# B&R Automation Studio project Laba2
Automation Studio 4.5.2.102

## Configuration labBR

CPU 4PP065.0571-P74, AutomationRuntime D4.52, Build 4.1.2, Vc V4.52.0, Safety 1.10

### Task classes (Cpu.sw)
```
Cyclic#1 (cycle 2000 us, tolerance 0 us):
  ncsdcctrl <- ncsdcctrl.prg
  DoorCtrl <- DoorCtrl.prg
Cyclic#7 (cycle 1000000 us, tolerance 1000000 us):
  LedCtrl <- LedCtrl.prg
DataObjects: Acp10sys, Arnc0sys
NcDataObjects: acp10etxen <- acp10etxen.dob, gmcipvar <- GmcIpUserConfig.gmcipvar.dob, gmcipfun <- GmcIpUserConfig.gmcipfun.dob, gmcipfub <- GmcIpUserConfig.gmcipfub.dob, gmcipubr <- GmcIpUserConfig.gmcipubr.dob, gmcipusm <- GmcIpUserConfig.gmcipusm.dob, gmcipui <- GmcIpUserConfig.gmcipui.dob, gmcipus <- GmcIpUserConfig.gmcipus.dob, gmcipuc <- GmcIpUserConfig.gmcipuc.dob, gmcipsys <- GmcIpConfig.gmcipsys.dob, gmciplbr <- GmcIpConfig.gmciplbr.dob, gmcipcbr <- GmcIpConfig.gmcipcbr.dob, gmciplsm <- GmcIpConfig.gmciplsm.dob, gmcipcsm <- GmcIpConfig.gmcipcsm.dob, gmcipcfg <- GmcIpConfig.gmcipcfg.dob, gmcipiec <- GmcIpConfig.gmcipiec.dob, gmciplog <- GmcIpConfig.gmciplog.dob, gmcipesm <- GmcIpConfig.gmcipesm.dob, gmcipmxd <- GmcIpConfig.gmcipmxd.dob, gmcipmx <- GmcIpConfig.gmcipmx.dob, gAxis01a <- gAxis01obj.gAxis01a.dob, gAxis01i <- gAxis01obj.gAxis01i.dob, gAxis02a <- gAxis02obj.gAxis02a.dob, gAxis02i <- gAxis02obj.gAxis02i.dob, gAxis03a <- gAxis03obj.gAxis03a.dob, gAxis03i <- gAxis03obj.gAxis03i.dob, gAxis04a <- gAxis04obj.gAxis04a.dob, gAxis04i <- gAxis04obj.gAxis04i.dob, gAxis05a <- gAxis05obj.gAxis05a.dob, gAxis05i <- gAxis05obj.gAxis05i.dob
Binaries: TCData, udbdef, iomap, sysconf, ashwac, ashwd, asfw, User, arconfig, Role, arnc0cfg, Arnc0map, Acp10map, acp10cfg
Libraries: Acp10man, Acp10par, NcGlobal, Acp10sdc, Arnc0man, DataObj, AsArLog, sys_lib, FileIO, AsArProf, AsMem, brsystem, runtime, astime, Acp10_MC, AsBrStr, X64Lib, GateCtrl, asieccon, powerlnk
```

### Hardware
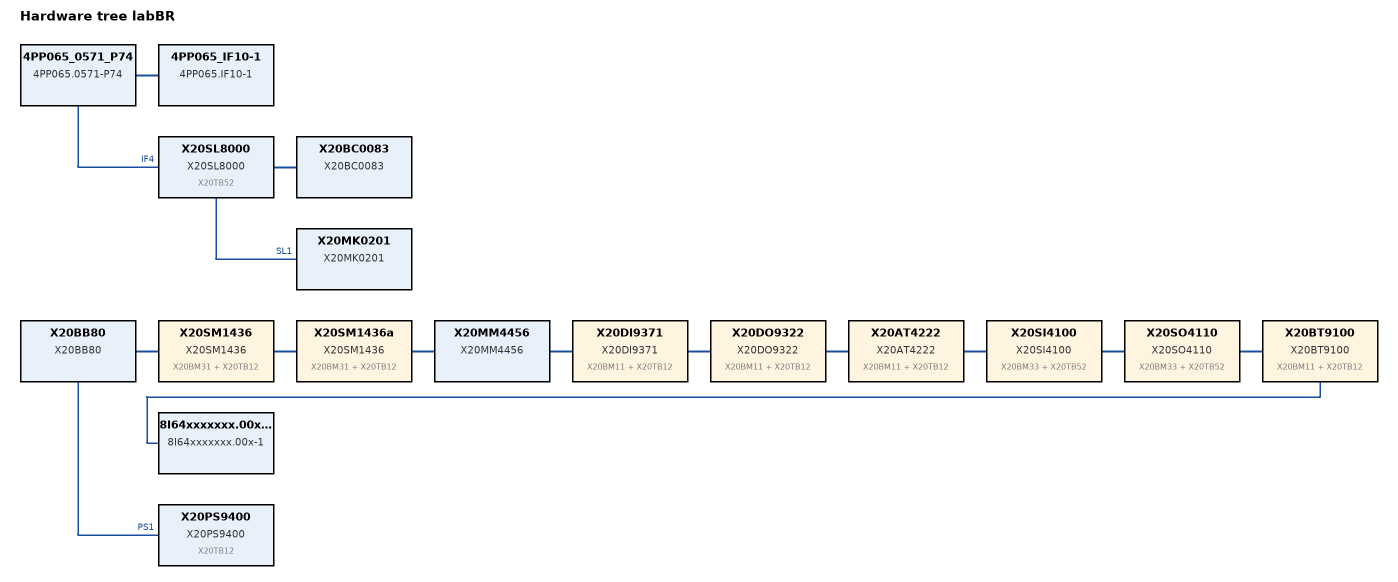
```
4PP065_0571_P74 : 4PP065.0571-P74 v1.1.2.0
  Connector IF4:
    EplInterfaceRedundant = 0
    EplEthInterfaceRedundant = 0
  Connector IF5:
    ActivateDevice = 1
    Mode = Manual
    InternetAddress = 10.1.1.13
    SubnetMask = 255.255.255.0
  ConfigurationID = DriveControl_SampleText
  TimerDeviceType = EPLX2X
  TimerDevice = 4PP065_0571_P74.IF4
  TaskClassIdleTime = 2000
  Cyclic1Duration = 2000
  Cyclic1Tolerance = 0
  Cyclic1Output = 1
  Cyclic2Duration = 20000
  Cyclic2Tolerance = 20000
  Cyclic3Duration = 50000
  Cyclic3Tolerance = 50000
  Cyclic4Duration = 100000
  Cyclic4Tolerance = 100000
  Cyclic5Duration = 200000
  Cyclic5Tolerance = 200000
  Cyclic6Duration = 500000
  Cyclic6Tolerance = 500000
  Cyclic7Duration = 1000000
  Cyclic7Tolerance = 1000000
  Cyclic8Duration = 10000
  Cyclic8Tolerance = 30000000
4PP065_IF10-1 : 4PP065.IF10-1 v1.0.3.0  [SS -> 4PP065_0571_P74.SS1]
8I64xxxxxxx.00x-1 : 8I64xxxxxxx.00x-1 v1.3.9.1  [X2X1 -> X20BT9100.X2X1 [Cable Type=X2XCable, Length=10, Version=1.0.0.2]]
  FunctionModel = Standard
  packedETAD = packed
  packedETI = packed
  packedCMDD = packed
  packedCMI = packed
  UNS = 220
  NCR = 10
  NSP = 890
  COS = 64
  RSC = 33000
X20AT4222 : X20AT4222 v1.2.3.0  [SS1 -> X20TB12e.SS; SL -> X20BM11c.SL1]
X20BB80 : X20BB80 v1.0.2.0
X20BC0083 : X20BC0083 v2.9.0.0  [PLK1 -> X20SL8000.PLK2 (NodeNumber=2) [Cable Type=PowerlinkCable, Length=10, Version=1.0.0.2]; SL -> X20BB80.SL1]
X20BM11 : X20BM11 v1.0.0.1  [X2X1 -> X20BM33a.X2X2]
X20BM11a : X20BM11 v1.0.0.1  [X2X1 -> X20MM4456.X2X2]
X20BM11b : X20BM11 v1.0.0.1  [X2X1 -> X20BM11a.X2X2]
X20BM11c : X20BM11 v1.0.0.1  [X2X1 -> X20BM11b.X2X2]
X20BM31 : X20BM31 v1.0.0.1  [X2X1 -> X20BB80.IF1]
X20BM31a : X20BM31 v1.0.0.1  [X2X1 -> X20BM31.X2X2]
X20BM33 : X20BM33 v1.0.0.4  [X2X1 -> X20BM11c.X2X2]
X20BM33a : X20BM33 v1.0.0.4  [X2X1 -> X20BM33.X2X2]
X20BT9100 : X20BT9100 v1.0.3.0  [SS1 -> X20TB12f.SS; SL -> X20BM11.SL1]
X20DI9371 : X20DI9371 v1.0.2.0  [SS1 -> X20TB12c.SS; SL -> X20BM11a.SL1]
X20DO9322 : X20DO9322 v1.0.3.0  [SS1 -> X20TB12d.SS; SL -> X20BM11b.SL1]
X20MK0201 : X20MK0201 v1.0.0.0  [SL -> X20SL8000.SL1]
X20MM4456 : X20MM4456 v1.1.5.0  [X2X1 -> X20BM31a.X2X2]
X20PS9400 : X20PS9400 v1.0.2.4  [SS1 -> X20TB12.SS; PS -> X20BB80.PS1]
X20SI4100 : X20SI4100 v1.10.1.1  [SS1 -> X20TB52.SS; SL -> X20BM33.SL1]
X20SL8000 : X20SL8000 v1.6.5.1  [PLK1 -> 4PP065_0571_P74.IF4 (NodeNumber=1) [Cable Type=PowerlinkCable, Length=10, Version=1.0.0.2]; PLK2 -> X20BC0083.PLK1 (NodeNumber=1) [Cable Type=PowerlinkCable, Length=10, Version=1.0.0.2]; SS1 -> X20TB52b.SS]
  SafeProject = SafeLOGIC-1
X20SM1436 : X20SM1436 v1.4.2.1  [SS1 -> X20TB12a.SS; SL -> X20BM31.SL1]
X20SM1436a : X20SM1436 v1.4.2.1  [SS1 -> X20TB12b.SS; SL -> X20BM31a.SL1]
X20SO4110 : X20SO4110 v1.10.1.1  [SS1 -> X20TB52a.SS; SL -> X20BM33a.SL1]
  SafeModuleID = 3
X20TB12 : X20TB12 v1.0.0.0
X20TB12a : X20TB12 v1.0.0.0
X20TB12b : X20TB12 v1.0.0.0
X20TB12c : X20TB12 v1.0.0.0
X20TB12d : X20TB12 v1.0.0.0
X20TB12e : X20TB12 v1.0.0.0
X20TB12f : X20TB12 v1.0.0.0
X20TB52 : X20TB52 v1.0.0.1
X20TB52a : X20TB52 v1.0.0.1
X20TB52b : X20TB52 v1.0.0.1
```

### IoMap.iom - 4PP065_0571_P74/IoMap.iom
```iecst
VAR_CONFIG
	::DoorCtrl:DoorBlock.s0 AT %IX."X20DI9371".DigitalInput02;
	::DoorCtrl:DoorBlock.s1 AT %IX."X20DI9371".DigitalInput03;
	::DoorCtrl:DoorBlock.s2 AT %IX."X20DI9371".DigitalInput04;
	::DoorCtrl:DoorBlock.s3 AT %IX."X20DI9371".DigitalInput05;
	::DoorCtrl:CMD AT %QW."8I64xxxxxxx.00x-1".CMDD_Output;
	::DoorCtrl:ETAD AT %IW."8I64xxxxxxx.00x-1".ETAD_Input;
	::DoorCtrl:Speed AT %QW."8I64xxxxxxx.00x-1".LFRD_Output;
END_VAR
```

## Logical view

Binary libraries used (declarations not repeated): operator, runtime, astime, AsIecCon, Acp10man, Acp10par, NcGlobal, Acp10sdc, Arnc0man, DataObj, AsArLog, sys_lib, FileIO, AsArProf, AsMem, brsystem, Acp10_MC, AsBrStr

### Global.var - Global variables
```iecst
VAR
	s1 : BOOL := FALSE;
	s2 : BOOL := FALSE;
	s3 : BOOL := FALSE;
	s0 : BOOL := FALSE;
END_VAR
```

### Package Logical/Libraries - Global libraries

### Library Logical/Libraries/X64Lib (ANSIC)

#### X64Lib.fun
```iecst
(********************************************************************
 * COPYRIGHT -- Microsoft
 ********************************************************************
 * Library: X64Lib
 * File: X64Lib.fun
 * Author: chuh
 * Created: April 02, 2015
 ********************************************************************
 * Functions and function blocks of library X64Lib
 ********************************************************************)

FUNCTION_BLOCK FBX64Inverter (*X64 Acopos Inverter Control Lib*) (*$GROUP=User*)
	VAR_INPUT
		enable : BOOL;
		ETAD_Input : UINT;
	END_VAR
	VAR_OUTPUT
		CMDD_Output : UINT;
	END_VAR
	VAR
		sex : UINT;
	END_VAR
END_FUNCTION_BLOCK
```

#### FBX64Inverter.c
```c
/********************************************************************
 * COPYRIGHT -- Microsoft
 ********************************************************************
 * Library: X64Lib
 * File: FBX64Inverter.c
 * Author: chuh
 * Created: April 02, 2015
 ********************************************************************
 * Implementation of library X64Lib
 ********************************************************************/

#include <bur/plctypes.h>
#ifdef __cplusplus
	extern "C"
	{
#endif

	#include "X64Lib.h"

#ifdef __cplusplus
	};
#endif

//***************Объявление списка состояний частотника ? ********************
#define	ACPIX64_STATE_NOT_READY_TO_SWITCH_ON	0x0000 /* */
#define	ACPIX64_STATE_SWITCH_ON_DISABLED		0x0040 /* */
#define	ACPIX64_STATE_READY_TO_SWITCH_ON		0x0064 /* */
#define	ACPIX64_STATE_SWITCHED_ON				0x0021 /* */
#define	ACPIX64_STATE_OPERATION_ENABLED			0x0027 /* */
#define	ACPIX64_STATE_QUICK_STOP_ACTIVE			0x0007/* */
#define	ACPIX64_STATE_MALFUNCTION				0x0008/* */

#define	ACPIX64_CMD_DISABLE_VOLTAGE				0x0000/* */
#define	ACPIX64_CMD_SHUTDOWN					0x0006/* */
#define	ACPIX64_CMD_SWITCH_ON					0x0006/* */
#define	ACPIX64_CMD_ENABLE_OPERATION			0x000F/* */
#define ACPIX64_CMD_GO                          0x0007
#define	ACPIX64_CMD_FAULT_RESET					0x0080/* */

/* X64 Acopos Inverter Control Lib */
void FBX64Inverter(struct FBX64Inverter* inst)
{
	UINT MSK;			//Переменная для хранения входа после наложения ма
	MSK = inst->ETAD_Input & 0x006F;
	inst->sex = MSK;/* */ // маска на значащую информацию статуса частотника
	if(!inst->enable){
		inst->CMDD_Output = ACPIX64_CMD_DISABLE_VOLTAGE;		//	 Отключаем питание с двигателя насоса
	} else {
		switch(MSK)
		{
			case ACPIX64_STATE_SWITCH_ON_DISABLED:		inst->CMDD_Output = ACPIX64_CMD_SHUTDOWN;				break;
			case ACPIX64_STATE_READY_TO_SWITCH_ON:		inst->CMDD_Output = ACPIX64_CMD_SWITCH_ON;				break;
			case ACPIX64_STATE_SWITCHED_ON:				inst->CMDD_Output = ACPIX64_CMD_ENABLE_OPERATION;		break;
		}
	}
}
```

### Library Logical/Libraries/GateCtrl (ANSIC)
Depends on: X64Lib

#### Types.typ - Exported data types
```iecst
TYPE
	GateState :
		(
		ST_INIT := 0,
		ST_UNKNOWN := 1,
		ST_OPEN := 2,
		ST_CLOSE := 3,
		ST_ACC_POS := 4,
		ST_NEG_ACC := 5,
		ST_POS := 6,
		ST_NEG := 7,
		ST_DEC_POS := 8,
		ST_DEC_NEG := 9
		);
END_TYPE
```

#### GateCtrl.fun - Exported functions and function blocks
```iecst
{REDUND_ERROR} FUNCTION_BLOCK FBGate (*СТЕПА САСИ*) (*$GROUP=User,$CAT=User,$GROUPICON=User.png,$CATICON=User.png*)
	VAR_INPUT
		s0 : BOOL; (*инпут датчиков*)
		s1 : BOOL;
		s2 : BOOL;
		s3 : BOOL;
	END_VAR
	VAR_OUTPUT
		S0 : BOOL; (*аутпут датчиков*)
		S1 : BOOL;
		S2 : BOOL;
		S3 : BOOL;
		Speed : INT;
	END_VAR
	VAR
		State : GateState;
		direction : USINT;
		DriveBlk : FBX64Inverter;
	END_VAR
END_FUNCTION_BLOCK
```

#### FBGate.c
```c
#include <bur/plctypes.h>
#ifdef __cplusplus
	extern "C"
	{
#endif
	#include "GateCtrl.h"
#ifdef __cplusplus
	};
#endif
/* TODO: Add your comment here */
void FBGate(struct FBGate* inst)
{
	switch (inst->State) {
		case ST_INIT: //Инициализация параметров и ожидание включения частотного преобразователя
			inst->State = ST_UNKNOWN;
			inst->S0 = 0;
			inst->S1 = 0;
			inst->S2 = 0;
			inst->S3 = 0;
			break;
		case ST_UNKNOWN: //Ворота в неизвестном положении
			if ((inst->direction == 0) && (inst->s0 == 0)){
			inst->State = ST_OPEN;
			}
			if ((inst->direction == 1) && (inst->s0 == 1)){
				inst->State = ST_CLOSE;
			}
			break;
		case ST_OPEN: //ворота открыты
			inst->DriveBlk.enable = 0;
			FBX64Inverter(&inst->DriveBlk);
			inst->S0 = 0;
			inst->S1 = 0;
			inst->S2 = 0;
			inst->S3 = 0;
			inst->Speed = 0;
			FBX64Inverter(&inst->DriveBlk);
			if (inst->direction == 1){
				inst->State = ST_ACC_POS;
			}
			break;
		case ST_CLOSE: //Ворота закрыты
			inst->DriveBlk.enable = 0;
			FBX64Inverter(&inst->DriveBlk);
			inst->S0 = 1;
			inst->S1 = 1;
			inst->S2 = 1;
			inst->S3 = 1;
			inst->Speed = 0;
			FBX64Inverter(&inst->DriveBlk);
			if (inst->direction == 0){
				inst->State = ST_NEG_ACC;
			}
			break;
		case ST_ACC_POS: //Ускорение ворот в строну открытия
			inst->DriveBlk.enable = 1;
			inst->S0 = 1;
			inst->S1 = 0;
			inst->S2 = 0;
			inst->S3 = 0;
			inst->Speed = 100;
			FBX64Inverter(&inst->DriveBlk);
			if (inst->s1){
				inst->State = ST_POS;
			}
			if (inst->direction == 0) {
				inst->State = ST_NEG_ACC;
			}
			break;
		case ST_NEG_ACC://Ускорение в строну закрытия
			inst->DriveBlk.enable = 1;
			FBX64Inverter(&inst->DriveBlk);
			inst->Speed = -100;
			inst->S0 = 1;
			inst->S1 = 1;
			inst->S2 = 1;
			inst->S3 = 0;
			if (inst->s2){
				inst->State = ST_NEG;
			}
			break;
		case ST_NEG: //Двиежние в сторону закрытия
			inst->Speed = -300;
			FBX64Inverter(&inst->DriveBlk);
			inst->S0 = 1;
			inst->S1 = 1;
			inst->S2 = 0;
			inst->S3 = 0;
			if (inst->s1){
				inst->State = ST_DEC_NEG;
			}

			break;
		case ST_DEC_NEG: //Замедление ворот в сторону закрытия
			inst->Speed = -100;
			FBX64Inverter(&inst->DriveBlk);
			inst->S0 = 1;
			inst->S1 = 0;
			inst->S2 = 0;
			inst->S3 = 0;
			if (inst->s0){
				inst->State = ST_OPEN;
			}
			break;
		case ST_DEC_POS: //Замедление ворот в сторону закрытия
			inst->S0 = 1;
			FBX64Inverter(&inst->DriveBlk);
			inst->S1 = 1;
			inst->S2 = 1;
			inst->S3 = 0;
			inst->Speed = 100;
			if (inst->s3){
				inst->State = ST_CLOSE;
			}
			break;
		case ST_POS: //Ускорение ворот в строну открытия
			inst->S0 = 1;
			FBX64Inverter(&inst->DriveBlk);
			inst->S1 = 1;
			inst->S2 = 0;
			inst->S3 = 0;
			inst->Speed = 300;
			if (inst->s2){
				inst->State = ST_DEC_POS;
			}
			if (inst->direction == 0) {
				inst->State = ST_NEG;
			}
			break;
	}
}
```

### Program Logical/DoorCtrl (ANSIC)

#### Variables.var
```iecst
VAR
	Close : BOOL;
	Open : BOOL;
	DoorBlock : FBGate;
	ETAD : UINT := 0;
	Speed : INT := 0;
	CMD : UINT := 0;
END_VAR
```

#### Main.c
```c
#include <bur/plctypes.h>

#ifdef _DEFAULT_INCLUDES
	#include <AsDefault.h>
#endif

void _INIT ProgramInit(void)
{
	Open  = 0;
	Close = 0;
}

void _CYCLIC ProgramCyclic(void)
{
	if (Open == 1){
		DoorBlock.direction = 1;
	}
	if (Close == 1) {
		DoorBlock.direction = 0;
	}
	FBGate(&DoorBlock);
	if ((DoorBlock.State == ST_OPEN) || (DoorBlock.State == ST_CLOSE)){
		Open  = 0;
		Close = 0;
	}
	s0 = DoorBlock.S0;
	s1 = DoorBlock.S1;
	s2 = DoorBlock.S2;
	s3 = DoorBlock.S3;

}

void _EXIT ProgramExit(void)
{

}
```

### Program Logical/LedCtrl (ANSIC)

#### Variables.var
```iecst
VAR
	sc0 : BOOL;
	sc1 : BOOL;
	sc2 : BOOL;
	sc3 : BOOL;
END_VAR
```

#### Main.c
```c
#include <bur/plctypes.h>

#ifdef _DEFAULT_INCLUDES
	#include <AsDefault.h>
#endif

void _INIT ProgramInit(void)
{

}

void _CYCLIC ProgramCyclic(void)
{
    if (s0 == 1)
		sc0 = !sc0;
	if (s1 == 1)
		sc1 = !sc1;
	if (s2 == 1)
		sc2 = !sc2;
	if (s3 == 1)
		sc3 = !sc3;
}

void _EXIT ProgramExit(void)
{

}
```

Listed in the project but not available here: Logical/Global.typ, Logical/Libraries/GateCtrl/Constants.var, Logical/ncsdcctrl, Logical/acp10etxen, Logical/GmcIpConfig, Logical/GmcIpUserConfig, Logical/gAxis01obj, Logical/gAxis02obj, Logical/gAxis03obj, Logical/gAxis04obj, Logical/gAxis05obj
